VAR_GLOBAL
	stGroupRef			: AXES_GROUP_REF;
	stAxis				: ARRAY[1..cAxesCount] OF AXIS_REF;
	stACSAxis			: ARRAY[1..cAxesCount] OF AXIS_REF;
	PointAPos			: ARRAY[1..5,1..9] OF MC_LREAL;
	PointAPos2			: ARRAY[1..5,1..6] OF MC_LREAL;
	PointBPos			: ARRAY[1..5,1..9] OF MC_LREAL;
	MidPointPos			: ARRAY[1..3] OF MC_LREAL;
	PointAMidPos		: ARRAY[1..3] OF MC_LREAL;
	PointBMidPos		: ARRAY[1..3] OF MC_LREAL;
	PointXTSMidPos		: ARRAY[1..3] OF MC_LREAL;
	PreviousUpPos		: ARRAY[1..3] OF MC_LREAL;
	DeltaVelocity		: INT := 200;
	UpToMidBlend		: INT := 0;
	MidToUpBlend		: INT := 0;
	PointXTSPos			: ARRAY[1..6] OF MC_LREAL;
END_VAR

VAR_GLOBAL CONSTANT
	cAxesCount			: UINT:=3;
END_VAR

(* stored: Version 1.1.0.1, ProductVersion 3.1.4024.6
   GVL GVL: Id {f09b62d0-c0a9-403a-804d-b72361a29bce} *)
